(* CoDeSys 2.3.9.55 project: CruceMoviles.pro *)
(* Libraries: Standard.lib 2.6.14 11:37:46 *)

(* Global variable list: Global_Variables *)
VAR_GLOBAL

      (*Entradas*)
      M1:BOOL;
      M2:BOOL;

	A1:BOOL;
	B1:BOOL;
       C1: BOOL;
       D1:BOOL;

	A2:BOOL;
	B2:BOOL;
      C2: BOOL;
       D2:BOOL;

       (* Salidas *)
	MOTOR_BA1:BOOL;
	MOTOR_FO1:BOOL;

       MOTOR_BA2:BOOL;
	MOTOR_FO2:BOOL;

      Carga1:BOOL;
      Carga2:BOOL;


      (* Variables del simulador *)
	Vel:INT:=1;
	Vel2:INT:=1;


END_VAR

(* POU PLC_PRG, ST *)
PROGRAM PLC_PRG
VAR
END_VAR
SimVehiculo;
SimVehiculo2;
Automatismo;
END_PROGRAM

(* POU SimVehiculo, ST *)
PROGRAM SimVehiculo
VAR
	PosX: INT;
END_VAR
A1:=FALSE;
B1:=FALSE;
C1:=FALSE;
D1:=FALSE;


IF MOTOR_FO1=TRUE THEN

     PosX:=PosX+Vel;

END_IF

IF MOTOR_BA1=TRUE THEN

     PosX:=PosX-Vel;

END_IF


IF PosX<=0 THEN
   A1:=TRUE;
END_IF

IF PosX>=129 AND   PosX<=199 THEN
   B1:=TRUE;
END_IF

IF PosX>=220 AND   PosX<=288 THEN
   C1:=TRUE;
END_IF

IF PosX>=438 THEN
  D1:=TRUE;
END_IF
END_PROGRAM

(* POU SimVehiculo2, ST *)
PROGRAM SimVehiculo2
VAR
	PosY2: INT;
END_VAR
A2:=FALSE;
B2:=FALSE;
C2:=FALSE;
D2:=FALSE;


IF MOTOR_FO2=TRUE THEN

     PosY2:=PosY2-Vel2;

END_IF

IF MOTOR_BA2=TRUE THEN

     PosY2:=PosY2+Vel2;

END_IF


IF PosY2>=0 THEN
   A2:=TRUE;
END_IF

IF PosY2<=-70 AND PosY2>=-142 THEN
  B2:=TRUE;
END_IF

IF PosY2<=-151 AND PosY2>=-220 THEN
  C2:=TRUE;
END_IF

IF PosY2<=-302  THEN
  D2:=TRUE;
END_IF
END_PROGRAM

(* POU Automatismo, LD *)
PROGRAM Automatismo
VAR

END_VAR
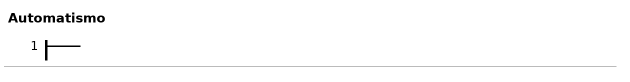
_LD_ (* Ladder Diagram *)
NETWORK 1
	*
_END_LD_
(* the same logic as Structured Text *)
(* Network 1 *)
END_PROGRAM

(* Visualisation Vehiculo
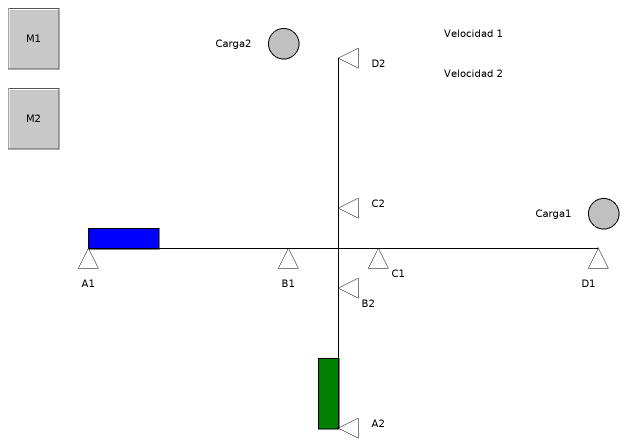
rectangle at (120,230)-(191,251): x offset SimVehiculo.PosX
polygon at (110,250)-(130,270): alarm colour if .A1
polygon at (620,250)-(640,270): alarm colour if .D1
button at (40,10)-(91,71): text "M1"; taps M1
rectangle at (350,360)-(371,431): y offset SimVehiculo2.PosY2
polygon at (370,420)-(390,440): alarm colour if .A2
rectangle at (450,20)-(561,51): text "Velocidad 1"
rectangle at (450,60)-(561,91): text "Velocidad 2"
polygon at (370,50)-(390,70): alarm colour if .D2
polygon at (310,250)-(330,270): alarm colour if .B1
polygon at (400,250)-(420,270): alarm colour if .C1
polygon at (370,280)-(390,300): alarm colour if .B2
polygon at (370,200)-(390,220): alarm colour if .C2
ellipse at (620,200)-(651,231): alarm colour if Carga1
rectangle at (530,200)-(641,231): text "Carga1"
ellipse at (300,30)-(331,61): alarm colour if Carga2
rectangle at (210,30)-(321,61): text "Carga2"
rectangle at (100,270)-(141,301): text "A1"
rectangle at (300,270)-(341,301): text "B1"
rectangle at (410,260)-(451,291): text "C1"
rectangle at (600,270)-(641,301): text "D1"
rectangle at (390,410)-(431,441): text "A2"
rectangle at (380,290)-(421,321): text "B2"
rectangle at (390,190)-(431,221): text "C2"
rectangle at (390,50)-(431,81): text "D2"
button at (40,90)-(91,151): text "M2"; taps M2
2 more shapes without text or variables
2 elements of other kinds (tables, trends, ...) not read
*)
